Yaskawa INFORM job: argaz_program.JBI

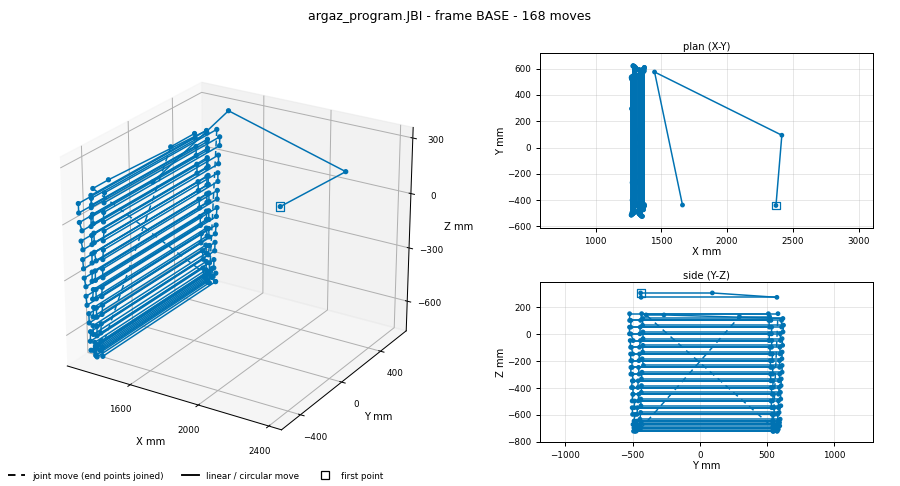
[picture p0: tool path of argaz_program.JBI in frame BASE, 168 of 174 moves have a stored position in this frame; points joined in program order, loops and branches not executed]
/JOB
//NAME ARGAZ_PROGRAM
//POS
///NPOS 168,0,168,0,0,0
///TOOL 0
///POSTYPE BASE
///RECTAN
///RCONF 0,0,0,0,0,0,0,0,0,0,0,0,0,0,0,0,0,0,0,0,0,0,0,0
C00000=2371.989878,-440.401884,308.020132,175.000000,5.000000,90.000000
C00001=2416.705806,93.738458,308.020132,175.000000,5.000000,90.000000
C00002=1448.862309,574.607175,275.381870,175.000000,5.000000,90.000000
C00003=1661.240590,-437.144282,275.381870,175.000000,5.000000,90.000000
C00004=1357.088440,511.287212,153.366162,175.000000,-89.999999,5.000000
C00005=1357.088440,-522.394236,153.366162,175.000000,-89.999999,5.000000
C00006=1354.164261,-522.287069,103.366162,175.000000,-89.999999,5.000000
C00007=1354.164261,514.938218,103.366162,175.000000,-89.999999,5.000000
C00008=1352.438438,518.625405,53.366162,175.000000,-89.999999,5.000000
C00009=1352.438438,-522.994646,53.366162,175.000000,-89.999999,5.000000
C00010=1350.832322,-523.178754,3.366162,175.000000,-89.999999,5.000000
C00011=1350.832322,518.871340,3.366162,175.000000,-89.999999,5.000000
C00012=1348.825152,516.219643,-46.633838,175.000000,-89.999999,5.000000
C00013=1348.825152,-518.107555,-46.633838,175.000000,-89.999999,5.000000
C00014=1347.044766,-514.870562,-96.633838,175.000000,-89.999999,5.000000
C00015=1347.044766,522.164664,-96.633838,175.000000,-89.999999,5.000000
C00016=1345.183955,525.111757,-146.633838,175.000000,-89.999999,5.000000
C00017=1345.183955,-515.018947,-146.633838,175.000000,-89.999999,5.000000
C00018=1343.293055,-513.493878,-196.633838,175.000000,-89.999999,5.000000
C00019=1343.293055,525.184576,-196.633838,175.000000,-89.999999,5.000000
C00020=1341.807234,528.689487,-246.633838,175.000000,-89.999999,5.000000
C00021=1341.807234,-512.923694,-246.633838,175.000000,-89.999999,5.000000
C00022=1339.870905,-513.256187,-296.633838,175.000000,-89.999999,5.000000
C00023=1339.870905,527.209758,-296.633838,175.000000,-89.999999,5.000000
C00024=1337.995986,529.873820,-346.633838,175.000000,-89.999999,5.000000
C00025=1337.995986,-502.334769,-346.633838,175.000000,-89.999999,5.000000
C00026=1336.213293,-508.248877,-396.633838,175.000000,-89.999999,5.000000
C00027=1336.213293,530.626737,-396.633838,175.000000,-89.999999,5.000000
C00028=1334.396229,540.131627,-446.633838,175.000000,-89.999999,5.000000
C00029=1334.396229,-499.231047,-446.633838,175.000000,-89.999999,5.000000
C00030=1332.129137,-503.451779,-496.633838,175.000000,-89.999999,5.000000
C00031=1332.129137,530.722913,-496.633838,175.000000,-89.999999,5.000000
C00032=1330.170759,536.350555,-546.633838,175.000000,-89.999999,5.000000
C00033=1330.170759,-503.270419,-546.633838,175.000000,-89.999999,5.000000
C00034=1328.250549,-500.170819,-596.633838,175.000000,-89.999999,5.000000
C00035=1328.250549,538.973399,-596.633838,175.000000,-89.999999,5.000000
C00036=1326.642116,540.301995,-646.633838,175.000000,-89.999999,5.000000
C00037=1326.642116,-487.964771,-646.633838,175.000000,-89.999999,5.000000
C00038=1324.806880,-489.352446,-696.633838,175.000000,-89.999999,5.000000
C00039=1324.806880,541.085139,-696.633838,175.000000,-89.999999,5.000000
C00040=1343.412797,545.195956,-671.633838,180.000000,-60.000000,0.000000
C00041=1343.412797,-497.251205,-671.633838,180.000000,-60.000000,0.000000
C00042=1342.156410,-493.079935,-721.633838,180.000000,-60.000000,0.000000
C00043=1342.156410,545.345715,-721.633838,180.000000,-60.000000,0.000000
C00044=1342.156410,545.345715,-721.633838,180.000000,-60.000000,0.000000
C00045=1371.377692,582.641704,153.649998,175.000000,-89.999999,5.000000
C00046=1371.377692,-432.613364,153.649998,175.000000,-89.999999,5.000000
C00047=1372.180185,-440.408458,103.649998,175.000000,-89.999999,5.000000
C00048=1372.180185,609.123405,103.649998,175.000000,-89.999999,5.000000
C00049=1371.089827,609.796808,53.649998,175.000000,-89.999999,5.000000
C00050=1371.089827,-443.667374,53.649998,175.000000,-89.999999,5.000000
C00051=1369.998045,-445.573285,3.649998,175.000000,-89.999999,5.000000
C00052=1369.998045,599.394857,3.649998,175.000000,-89.999999,5.000000
C00053=1369.110863,601.830265,-46.350002,175.000000,-89.999999,5.000000
C00054=1369.110863,-441.873008,-46.350002,175.000000,-89.999999,5.000000
C00055=1367.639331,-448.976108,-96.350002,175.000000,-89.999999,5.000000
C00056=1367.639331,596.630322,-96.350002,175.000000,-89.999999,5.000000
C00057=1366.582076,598.500428,-146.350002,175.000000,-89.999999,5.000000
C00058=1366.582076,-448.746131,-146.350002,175.000000,-89.999999,5.000000
C00059=1365.085299,-453.213455,-196.350002,175.000000,-89.999999,5.000000
C00060=1365.085299,594.650047,-196.350002,175.000000,-89.999999,5.000000
C00061=1363.658730,594.990191,-246.350002,175.000000,-89.999999,5.000000
C00062=1363.658730,-455.754211,-246.350002,175.000000,-89.999999,5.000000
C00063=1361.864342,-451.909338,-296.350002,175.000000,-89.999999,5.000000
C00064=1361.864342,595.571329,-296.350002,175.000000,-89.999999,5.000000
C00065=1360.073877,591.872429,-346.350002,175.000000,-89.999999,5.000000
C00066=1360.073877,-458.655768,-346.350002,175.000000,-89.999999,5.000000
C00067=1358.161888,-460.748966,-396.350002,175.000000,-89.999999,5.000000
C00068=1358.161888,591.928890,-396.350002,175.000000,-89.999999,5.000000
C00069=1356.405837,587.009877,-446.350002,175.000000,-89.999999,5.000000
C00070=1356.405837,-453.709213,-446.350002,175.000000,-89.999999,5.000000
C00071=1354.608405,-458.341789,-496.350002,175.000000,-89.999999,5.000000
C00072=1354.608405,586.376409,-496.350002,175.000000,-89.999999,5.000000
C00073=1352.468508,585.807665,-546.350002,175.000000,-89.999999,5.000000
C00074=1352.468508,-463.981028,-546.350002,175.000000,-89.999999,5.000000
C00075=1350.405576,-467.600056,-596.350002,175.000000,-89.999999,5.000000
C00076=1350.405576,580.519588,-596.350002,175.000000,-89.999999,5.000000
C00077=1348.479511,582.258869,-646.350002,175.000000,-89.999999,5.000000
C00078=1348.479511,-467.412770,-646.350002,175.000000,-89.999999,5.000000
C00079=1346.462576,-469.588593,-696.350002,175.000000,-89.999999,5.000000
C00080=1346.462576,577.739216,-696.350002,175.000000,-89.999999,5.000000
C00081=1364.869259,576.218205,-671.350002,180.000000,-60.000000,0.000000
C00082=1364.869259,-472.867477,-671.350002,180.000000,-60.000000,0.000000
C00083=1363.104675,-472.908790,-721.350002,180.000000,-60.000000,0.000000
C00084=1363.104675,576.344210,-721.350002,180.000000,-60.000000,0.000000
C00085=1363.104675,576.344210,-721.350002,180.000000,-60.000000,0.000000
C00086=1277.888245,-399.618923,144.199188,175.000000,-89.999999,5.000000
C00087=1277.888245,-266.558107,144.199188,175.000000,-89.999999,5.000000
C00088=1283.410944,619.398505,117.816493,175.000000,-89.999999,5.000000
C00089=1283.410944,-424.812790,117.816493,175.000000,-89.999999,5.000000
C00090=1286.253415,-425.480523,67.816493,175.000000,-89.999999,5.000000
C00091=1286.253415,623.737395,67.816493,175.000000,-89.999999,5.000000
C00092=1288.733474,620.101960,17.816493,175.000000,-89.999999,5.000000
C00093=1288.733474,-423.231390,17.816493,175.000000,-89.999999,5.000000
C00094=1291.050491,-422.345201,-32.183507,175.000000,-89.999999,5.000000
C00095=1291.050491,613.233653,-32.183507,175.000000,-89.999999,5.000000
C00096=1293.592039,617.319739,-82.183507,175.000000,-89.999999,5.000000
C00097=1293.592039,-423.386645,-82.183507,175.000000,-89.999999,5.000000
C00098=1295.614737,-424.881487,-132.183507,175.000000,-89.999999,5.000000
C00099=1295.614737,613.520806,-132.183507,175.000000,-89.999999,5.000000
C00100=1297.247512,612.008789,-182.183507,175.000000,-89.999999,5.000000
C00101=1297.247512,-429.228621,-182.183507,175.000000,-89.999999,5.000000
C00102=1299.433219,-419.216748,-232.183507,175.000000,-89.999999,5.000000
C00103=1299.433219,613.471344,-232.183507,175.000000,-89.999999,5.000000
C00104=1300.418371,613.420508,-282.183507,175.000000,-89.999999,5.000000
C00105=1300.418371,-430.256325,-282.183507,175.000000,-89.999999,5.000000
C00106=1302.234326,-433.734445,-332.183507,175.000000,-89.999999,5.000000
C00107=1302.234326,606.925912,-332.183507,175.000000,-89.999999,5.000000
C00108=1303.707506,605.868668,-382.183507,175.000000,-89.999999,5.000000
C00109=1303.707506,-433.869777,-382.183507,175.000000,-89.999999,5.000000
C00110=1305.086846,-435.019762,-432.183507,175.000000,-89.999999,5.000000
C00111=1305.086846,600.756939,-432.183507,175.000000,-89.999999,5.000000
C00112=1306.071877,603.429245,-482.183507,175.000000,-89.999999,5.000000
C00113=1306.071877,-438.802208,-482.183507,175.000000,-89.999999,5.000000
C00114=1307.412042,-438.117988,-532.183507,175.000000,-89.999999,5.000000
C00115=1307.412042,603.875774,-532.183507,175.000000,-89.999999,5.000000
C00116=1308.466459,591.089237,-582.183507,175.000000,-89.999999,5.000000
C00117=1308.466459,-439.996158,-582.183507,175.000000,-89.999999,5.000000
C00118=1310.304432,-445.204750,-632.183507,175.000000,-89.999999,5.000000
C00119=1310.304432,598.888386,-632.183507,175.000000,-89.999999,5.000000
C00120=1311.312316,595.813517,-682.183507,175.000000,-89.999999,5.000000
C00121=1311.312316,-443.494887,-682.183507,175.000000,-89.999999,5.000000
C00122=1332.658786,-435.818706,-657.183507,180.000000,-60.000000,0.000000
C00123=1332.658786,594.168915,-657.183507,180.000000,-60.000000,0.000000
C00124=1333.118383,585.110554,-707.183507,180.000000,-60.000000,0.000000
C00125=1333.118383,-444.618080,-707.183507,180.000000,-60.000000,0.000000
C00126=1333.118383,-444.618080,-707.183507,180.000000,-60.000000,0.000000
C00127=1273.288256,295.502746,131.277012,175.000000,-89.999999,5.000000
C00128=1273.288256,520.035994,131.277012,175.000000,-89.999999,5.000000
C00129=1270.890439,529.755591,103.296988,175.000000,-89.999999,5.000000
C00130=1270.890439,-513.266015,103.296988,175.000000,-89.999999,5.000000
C00131=1271.533657,-513.209554,53.296988,175.000000,-89.999999,5.000000
C00132=1271.533657,535.502244,53.296988,175.000000,-89.999999,5.000000
C00133=1273.366070,534.257342,3.296988,175.000000,-89.999999,5.000000
C00134=1273.366070,-513.096632,3.296988,175.000000,-89.999999,5.000000
C00135=1275.404717,-495.948939,-46.703012,175.000000,-89.999999,5.000000
C00136=1275.404717,536.502021,-46.703012,175.000000,-89.999999,5.000000
C00137=1277.028835,534.815069,-96.703012,175.000000,-89.999999,5.000000
C00138=1277.028835,-508.386938,-96.703012,175.000000,-89.999999,5.000000
C00139=1279.183844,-498.977189,-146.703012,175.000000,-89.999999,5.000000
C00140=1279.183844,540.662251,-146.703012,175.000000,-89.999999,5.000000
C00141=1280.966410,539.787790,-196.703012,175.000000,-89.999999,5.000000
C00142=1280.966410,-505.503283,-196.703012,175.000000,-89.999999,5.000000
C00143=1282.925389,-503.396314,-246.703012,175.000000,-89.999999,5.000000
C00144=1282.925389,542.645280,-246.703012,175.000000,-89.999999,5.000000
C00145=1285.047149,543.565873,-296.703012,175.000000,-89.999999,5.000000
C00146=1285.047149,-503.499597,-296.703012,175.000000,-89.999999,5.000000
C00147=1287.369843,-494.427239,-346.703012,175.000000,-89.999999,5.000000
C00148=1287.369843,546.345557,-346.703012,175.000000,-89.999999,5.000000
C00149=1289.521115,543.757979,-396.703012,175.000000,-89.999999,5.000000
C00150=1289.521115,-498.930368,-396.703012,175.000000,-89.999999,5.000000
C00151=1291.635581,-495.764407,-446.703012,175.000000,-89.999999,5.000000
C00152=1291.635581,549.175964,-446.703012,175.000000,-89.999999,5.000000
C00153=1293.849911,541.736391,-496.703012,175.000000,-89.999999,5.000000
C00154=1293.849911,-485.793718,-496.703012,175.000000,-89.999999,5.000000
C00155=1295.977049,-487.912163,-546.703012,175.000000,-89.999999,5.000000
C00156=1295.977049,552.744957,-546.703012,175.000000,-89.999999,5.000000
C00157=1298.303918,555.349060,-596.703012,175.000000,-89.999999,5.000000
C00158=1298.303918,-482.618577,-596.703012,175.000000,-89.999999,5.000000
C00159=1300.270344,-489.107488,-646.703012,175.000000,-89.999999,5.000000
C00160=1300.270344,549.567979,-646.703012,175.000000,-89.999999,5.000000
C00161=1302.656383,551.655668,-696.703012,175.000000,-89.999999,5.000000
C00162=1302.656383,-488.761835,-696.703012,175.000000,-89.999999,5.000000
C00163=1324.870088,-481.376429,-671.703012,180.000000,-60.000000,0.000000
C00164=1324.870088,551.349951,-671.703012,180.000000,-60.000000,0.000000
C00165=1327.105759,551.261816,-721.703012,180.000000,-60.000000,0.000000
C00166=1327.105759,-481.969961,-721.703012,180.000000,-60.000000,0.000000
C00167=1327.105759,-481.969961,-721.703012,180.000000,-60.000000,0.000000
///POSTYPE PULSE
///PULSE
EC00000=0
EC00001=0
EC00002=0
EC00003=0
EC00004=0
EC00005=0
EC00006=0
EC00007=0
EC00008=0
EC00009=0
EC00010=0
EC00011=0
EC00012=0
EC00013=0
EC00014=0
EC00015=0
EC00016=0
EC00017=0
EC00018=0
EC00019=0
EC00020=0
EC00021=0
EC00022=0
EC00023=0
EC00024=0
EC00025=0
EC00026=0
EC00027=0
EC00028=0
EC00029=0
EC00030=0
EC00031=0
EC00032=0
EC00033=0
EC00034=0
EC00035=0
EC00036=0
EC00037=0
EC00038=0
EC00039=0
EC00040=0
EC00041=0
EC00042=0
EC00043=0
EC00044=92160
EC00045=92160
EC00046=92160
EC00047=92160
EC00048=92160
EC00049=92160
EC00050=92160
EC00051=92160
EC00052=92160
EC00053=92160
EC00054=92160
EC00055=92160
EC00056=92160
EC00057=92160
EC00058=92160
EC00059=92160
EC00060=92160
EC00061=92160
EC00062=92160
EC00063=92160
EC00064=92160
EC00065=92160
EC00066=92160
EC00067=92160
EC00068=92160
EC00069=92160
EC00070=92160
EC00071=92160
EC00072=92160
EC00073=92160
EC00074=92160
EC00075=92160
EC00076=92160
EC00077=92160
EC00078=92160
EC00079=92160
EC00080=92160
EC00081=92160
EC00082=92160
EC00083=92160
EC00084=92160
EC00085=184320
EC00086=184320
EC00087=184320
EC00088=184320
EC00089=184320
EC00090=184320
EC00091=184320
EC00092=184320
EC00093=184320
EC00094=184320
EC00095=184320
EC00096=184320
EC00097=184320
EC00098=184320
EC00099=184320
EC00100=184320
EC00101=184320
EC00102=184320
EC00103=184320
EC00104=184320
EC00105=184320
EC00106=184320
EC00107=184320
EC00108=184320
EC00109=184320
EC00110=184320
EC00111=184320
EC00112=184320
EC00113=184320
EC00114=184320
EC00115=184320
EC00116=184320
EC00117=184320
EC00118=184320
EC00119=184320
EC00120=184320
EC00121=184320
EC00122=184320
EC00123=184320
EC00124=184320
EC00125=184320
EC00126=276480
EC00127=276480
EC00128=276480
EC00129=276480
EC00130=276480
EC00131=276480
EC00132=276480
EC00133=276480
EC00134=276480
EC00135=276480
EC00136=276480
EC00137=276480
EC00138=276480
EC00139=276480
EC00140=276480
EC00141=276480
EC00142=276480
EC00143=276480
EC00144=276480
EC00145=276480
EC00146=276480
EC00147=276480
EC00148=276480
EC00149=276480
EC00150=276480
EC00151=276480
EC00152=276480
EC00153=276480
EC00154=276480
EC00155=276480
EC00156=276480
EC00157=276480
EC00158=276480
EC00159=276480
EC00160=276480
EC00161=276480
EC00162=276480
EC00163=276480
EC00164=276480
EC00165=276480
EC00166=276480
EC00167=368640
//INST
///DATE 2023/01/29 12:01
///ATTR SC,RW,RJ
////FRAME BASE
///GROUP1 RB1,ST1
NOP
MOVJ P009 EX000 VJ=15.00
MOVJ C00000 EC00000 VJ=15.0
CALL JOB:SPYON
MOVL C00001 EC00001 V=150.0
MOVL C00002 EC00002 V=150.0
MOVL C00003 EC00003 V=150.0
CALL JOB:SPYOF
MOVJ P009 VJ=15.00
MOVJ C00004 EC00004 VJ=15.0
CALL JOB:SPYON
MOVL C00005 EC00005 V=150.0
MOVL C00006 EC00006 V=150.0
MOVL C00007 EC00007 V=150.0
MOVL C00008 EC00008 V=150.0
MOVL C00009 EC00009 V=150.0
MOVL C00010 EC00010 V=150.0
MOVL C00011 EC00011 V=150.0
MOVL C00012 EC00012 V=150.0
MOVL C00013 EC00013 V=150.0
MOVL C00014 EC00014 V=150.0
MOVL C00015 EC00015 V=150.0
MOVL C00016 EC00016 V=150.0
MOVL C00017 EC00017 V=150.0
MOVL C00018 EC00018 V=150.0
MOVL C00019 EC00019 V=150.0
MOVL C00020 EC00020 V=150.0
MOVL C00021 EC00021 V=150.0
MOVL C00022 EC00022 V=150.0
MOVL C00023 EC00023 V=150.0
MOVL C00024 EC00024 V=150.0
MOVL C00025 EC00025 V=150.0
MOVL C00026 EC00026 V=150.0
MOVL C00027 EC00027 V=150.0
MOVL C00028 EC00028 V=150.0
MOVL C00029 EC00029 V=150.0
MOVL C00030 EC00030 V=150.0
MOVL C00031 EC00031 V=150.0
MOVL C00032 EC00032 V=150.0
MOVL C00033 EC00033 V=150.0
MOVL C00034 EC00034 V=150.0
MOVL C00035 EC00035 V=150.0
MOVL C00036 EC00036 V=150.0
MOVL C00037 EC00037 V=150.0
MOVL C00038 EC00038 V=150.0
MOVL C00039 EC00039 V=150.0
MOVL C00040 EC00040 V=150.0
MOVL C00041 EC00041 V=150.0
MOVL C00042 EC00042 V=150.0
MOVL C00043 EC00043 V=150.0
CALL JOB:SPYOF
MOVJ P009 VJ=15.00
MOVL C00044 EC00044 V=150.0
MOVJ C00045 EC00045 VJ=15.0
CALL JOB:SPYON
MOVL C00046 EC00046 V=150.0
MOVL C00047 EC00047 V=150.0
MOVL C00048 EC00048 V=150.0
MOVL C00049 EC00049 V=150.0
MOVL C00050 EC00050 V=150.0
MOVL C00051 EC00051 V=150.0
MOVL C00052 EC00052 V=150.0
MOVL C00053 EC00053 V=150.0
MOVL C00054 EC00054 V=150.0
MOVL C00055 EC00055 V=150.0
MOVL C00056 EC00056 V=150.0
MOVL C00057 EC00057 V=150.0
MOVL C00058 EC00058 V=150.0
MOVL C00059 EC00059 V=150.0
MOVL C00060 EC00060 V=150.0
MOVL C00061 EC00061 V=150.0
MOVL C00062 EC00062 V=150.0
MOVL C00063 EC00063 V=150.0
MOVL C00064 EC00064 V=150.0
MOVL C00065 EC00065 V=150.0
MOVL C00066 EC00066 V=150.0
MOVL C00067 EC00067 V=150.0
MOVL C00068 EC00068 V=150.0
MOVL C00069 EC00069 V=150.0
MOVL C00070 EC00070 V=150.0
MOVL C00071 EC00071 V=150.0
MOVL C00072 EC00072 V=150.0
MOVL C00073 EC00073 V=150.0
MOVL C00074 EC00074 V=150.0
MOVL C00075 EC00075 V=150.0
MOVL C00076 EC00076 V=150.0
MOVL C00077 EC00077 V=150.0
MOVL C00078 EC00078 V=150.0
MOVL C00079 EC00079 V=150.0
MOVL C00080 EC00080 V=150.0
MOVL C00081 EC00081 V=150.0
MOVL C00082 EC00082 V=150.0
MOVL C00083 EC00083 V=150.0
MOVL C00084 EC00084 V=150.0
CALL JOB:SPYOF
MOVJ P009 VJ=15.00
MOVL C00085 EC00085 V=150.0
MOVJ C00086 EC00086 VJ=15.0
CALL JOB:SPYON
MOVL C00087 EC00087 V=150.0
MOVL C00088 EC00088 V=150.0
MOVL C00089 EC00089 V=150.0
MOVL C00090 EC00090 V=150.0
MOVL C00091 EC00091 V=150.0
MOVL C00092 EC00092 V=150.0
MOVL C00093 EC00093 V=150.0
MOVL C00094 EC00094 V=150.0
MOVL C00095 EC00095 V=150.0
MOVL C00096 EC00096 V=150.0
MOVL C00097 EC00097 V=150.0
MOVL C00098 EC00098 V=150.0
MOVL C00099 EC00099 V=150.0
MOVL C00100 EC00100 V=150.0
MOVL C00101 EC00101 V=150.0
MOVL C00102 EC00102 V=150.0
MOVL C00103 EC00103 V=150.0
MOVL C00104 EC00104 V=150.0
MOVL C00105 EC00105 V=150.0
MOVL C00106 EC00106 V=150.0
MOVL C00107 EC00107 V=150.0
MOVL C00108 EC00108 V=150.0
MOVL C00109 EC00109 V=150.0
MOVL C00110 EC00110 V=150.0
MOVL C00111 EC00111 V=150.0
MOVL C00112 EC00112 V=150.0
MOVL C00113 EC00113 V=150.0
MOVL C00114 EC00114 V=150.0
MOVL C00115 EC00115 V=150.0
MOVL C00116 EC00116 V=150.0
MOVL C00117 EC00117 V=150.0
MOVL C00118 EC00118 V=150.0
MOVL C00119 EC00119 V=150.0
MOVL C00120 EC00120 V=150.0
MOVL C00121 EC00121 V=150.0
MOVL C00122 EC00122 V=150.0
MOVL C00123 EC00123 V=150.0
MOVL C00124 EC00124 V=150.0
MOVL C00125 EC00125 V=150.0
CALL JOB:SPYOF
MOVJ P009 VJ=15.00
MOVL C00126 EC00126 V=150.0
MOVJ C00127 EC00127 VJ=15.0
CALL JOB:SPYON
MOVL C00128 EC00128 V=150.0
MOVL C00129 EC00129 V=150.0
MOVL C00130 EC00130 V=150.0
MOVL C00131 EC00131 V=150.0
MOVL C00132 EC00132 V=150.0
MOVL C00133 EC00133 V=150.0
MOVL C00134 EC00134 V=150.0
MOVL C00135 EC00135 V=150.0
MOVL C00136 EC00136 V=150.0
MOVL C00137 EC00137 V=150.0
MOVL C00138 EC00138 V=150.0
MOVL C00139 EC00139 V=150.0
MOVL C00140 EC00140 V=150.0
MOVL C00141 EC00141 V=150.0
MOVL C00142 EC00142 V=150.0
MOVL C00143 EC00143 V=150.0
MOVL C00144 EC00144 V=150.0
MOVL C00145 EC00145 V=150.0
MOVL C00146 EC00146 V=150.0
MOVL C00147 EC00147 V=150.0
MOVL C00148 EC00148 V=150.0
MOVL C00149 EC00149 V=150.0
MOVL C00150 EC00150 V=150.0
MOVL C00151 EC00151 V=150.0
MOVL C00152 EC00152 V=150.0
MOVL C00153 EC00153 V=150.0
MOVL C00154 EC00154 V=150.0
MOVL C00155 EC00155 V=150.0
MOVL C00156 EC00156 V=150.0
MOVL C00157 EC00157 V=150.0
MOVL C00158 EC00158 V=150.0
MOVL C00159 EC00159 V=150.0
MOVL C00160 EC00160 V=150.0
MOVL C00161 EC00161 V=150.0
MOVL C00162 EC00162 V=150.0
MOVL C00163 EC00163 V=150.0
MOVL C00164 EC00164 V=150.0
MOVL C00165 EC00165 V=150.0
MOVL C00166 EC00166 V=150.0
CALL JOB:SPYOF
MOVJ P009 VJ=15.00
MOVL C00167 EC00167 V=150.0
END
